(* CoDeSys 2.3 export: SETTINGS.EXP *)

(* Global variable list: Settings *)
VAR_GLOBAL RETAIN
	K14UZSPumpSpeed : USINT := 100;
END_VAR
